// TwinCAT 3 PLC project PLCInterpolation
// libraries:
//   TC2_Converted,1.1.0.0,aaaa
//   Tc2_Math, * (Beckhoff Automation GmbH)
//   Tc2_NC, * (Beckhoff Automation GmbH)
//   Tc2_NCI, * (Beckhoff Automation GmbH)
//   Tc2_PlcInterpolation, * (Beckhoff Automation GmbH)
//   Tc2_Standard, * (Beckhoff Automation GmbH)
//   Tc2_System, * (Beckhoff Automation GmbH)
//   Tc2_Utilities, * (Beckhoff Automation GmbH)
//   Tc3_Module, * (Beckhoff Automation GmbH)
// project tree:
//   Data types/ E_ACTIONTYPE.TcDUT, E_CONTROL_MODE.TcDUT, E_PROGRAM_STATE.TcDUT, ST_EXECUTION_TABLE.TcDUT, ST_PROGRAM.TcDUT
//   Global Variables/ Global_Variables.TcGVL, PROGRAMS.TcGVL, SETTINGS.TcGVL, TwinCAT_Import.TcGVL, Variable_Configuration.TcGVL
//   POUs/ FB_AxisEnable.TcPOU, FB_ChannelReset.TcPOU, FB_ChannelStartStop.TcPOU, FB_Execute.TcPOU, FB_SelectProgram.TcPOU, MAIN.TcPOU
//   / Standard.TcTTO

CONFIGURATION PLCInterpolation
    RESOURCE PLC ON TwinCAT3
        TASK Standard(INTERVAL := T#10ms, PRIORITY := 22);
        PROGRAM MAIN WITH Standard : MAIN;
    END_RESOURCE
END_CONFIGURATION

// ---- Data types/E_ACTIONTYPE.TcDUT
TYPE E_ACTIONTYPE :
(
	NONE,
	MOVE_X,
	MOVE_Y,
	MOVE_XY,
	MOVE_CIRCULAR,
	HOME,
	END
);
END_TYPE

// ---- Data types/E_CONTROL_MODE.TcDUT
TYPE E_CONTROL_MODE :
(
	E_REF_MODE,
	E_JOG_MODE,
	E_AUTO_MODE
);
END_TYPE

// ---- Data types/E_PROGRAM_STATE.TcDUT
TYPE E_PROGRAM_STATE :
(
	E_PROGRAMSTATE_NONE,
	E_PROGRAMSTATE_READY,
	E_PROGRAMSTATE_RESETTED,
	E_PROGRAMSTATE_RUNNING,
	E_PROGRAMSTATE_STOPPED,
	E_PROGRAMSTATE_ERROR
);
END_TYPE

// ---- Data types/ST_EXECUTION_TABLE.TcDUT
TYPE ST_EXECUTION_TABLE :
STRUCT
	ActionType:E_ACTIONTYPE;
	X:LREAL;
	Y:LREAL;
	I:LREAL;
	J:LREAL;
	Clockwise:BOOL;
END_STRUCT
END_TYPE

// ---- Data types/ST_PROGRAM.TcDUT
TYPE ST_PROGRAM :
STRUCT
	Name:STRING;
	Comment:STRING;
	ExecutionTable:ARRAY[1..MAX_NUMBER_OF_TABLE_LINES] OF ST_EXECUTION_TABLE;
END_STRUCT
END_TYPE

// ---- Global Variables/Global_Variables.TcGVL
{attribute 'Tc2GvlVarNames'}
VAR_GLOBAL
	in_stXNcToPlc		AT %I*:	NCTOPLC_AXIS_REF;
	in_stYNcToPlc		AT %I*:	NCTOPLC_AXIS_REF;
	in_stZNcToPlc		AT %I*:	NCTOPLC_AXIS_REF;

	in_stItpToPlc		AT %I*:	NCTOPLC_NCICHANNEL_REF;


	out_stXPlcToNc		AT	%Q*:	PLCTONC_AXIS_REF;
	out_stYPlcToNc		AT	%Q*:	PLCTONC_AXIS_REF;
	out_stZPlcToNc		AT	%Q*:	PLCTONC_AXIS_REF;

	out_stPlcToItp		AT	%Q*:	PLCTONC_NCICHANNEL_REF;


	gGlobalEnable: BOOL:=TRUE;
	gFeedOverride:	LREAL	:= 100.0;
	gVelocity: UINT:=1000;

	gControlMode:E_CONTROL_MODE:=E_AUTO_MODE;			(* Defines is control in REF, JOG or AUTO mode *)
	gProgramState: E_PROGRAM_STATE;		(* Defines status of the current program *)
	gStatistics_LastProgramTime:REAL; (* Last program time in seconds *)


	(* Visualization variables *)
	gVisuStart:BOOL;
	gVisuStop:BOOL;
	gVisuReset:BOOL;

	gVisuPrgNumber: INT;
	gVisuSelectPrg: BOOL;

END_VAR

VAR_GLOBAL CONSTANT
	ItpChnId:	UDINT := 2;
	ItpGrpId:	UDINT := 4;

	MAX_NUMBER_OF_TABLE_LINES:UINT:=100;
	MAX_NUMBER_OF_PROGRAMS:UINT:=10;

END_VAR

// ---- Global Variables/PROGRAMS.TcGVL
{attribute 'Tc2GvlVarNames'}
VAR_GLOBAL PERSISTENT
	gPrograms:ARRAY[1..MAX_NUMBER_OF_PROGRAMS] OF ST_PROGRAM;
	gCurrentProgram:ST_PROGRAM;
	giProgramNumber:INT;
END_VAR

// ---- Global Variables/SETTINGS.TcGVL
{attribute 'Tc2GvlVarNames'}
VAR_GLOBAL PERSISTENT
	(* Axis reference positions *)
	X_REF:LREAL:=0;
	Y_REF:LREAL:=0;

	(* Home position for axis *)
	X_Home:LREAL:=0;
	Y_Home:LREAL:=0;

END_VAR

// ---- Global Variables/TwinCAT_Import.TcGVL
{attribute 'Tc2GvlVarNames'}
(* Generated automatically by TwinCAT - do not edit manually! *)
VAR_GLOBAL
END_VAR

// ---- Global Variables/Variable_Configuration.TcGVL
{attribute 'Tc2GvlVarNames'}
VAR_CONFIG
END_VAR

// ---- POUs/MAIN.TcPOU
PROGRAM MAIN
VAR
	fbBuilGroup: CfgBuildExt3DGroup;
	fbExecute: FB_Execute;
	fbChannelReset: FB_ChannelReset;

	fbStartStop: FB_ChannelStartStop;
	rtSlideStart:R_TRIG;

	tmrReset: TON;

	fbSelectPrg: FB_SelectProgram;

	fbReleaseGroup: CfgReconfigGroup;

	fbEnable: FB_AxisEnable;
END_VAR

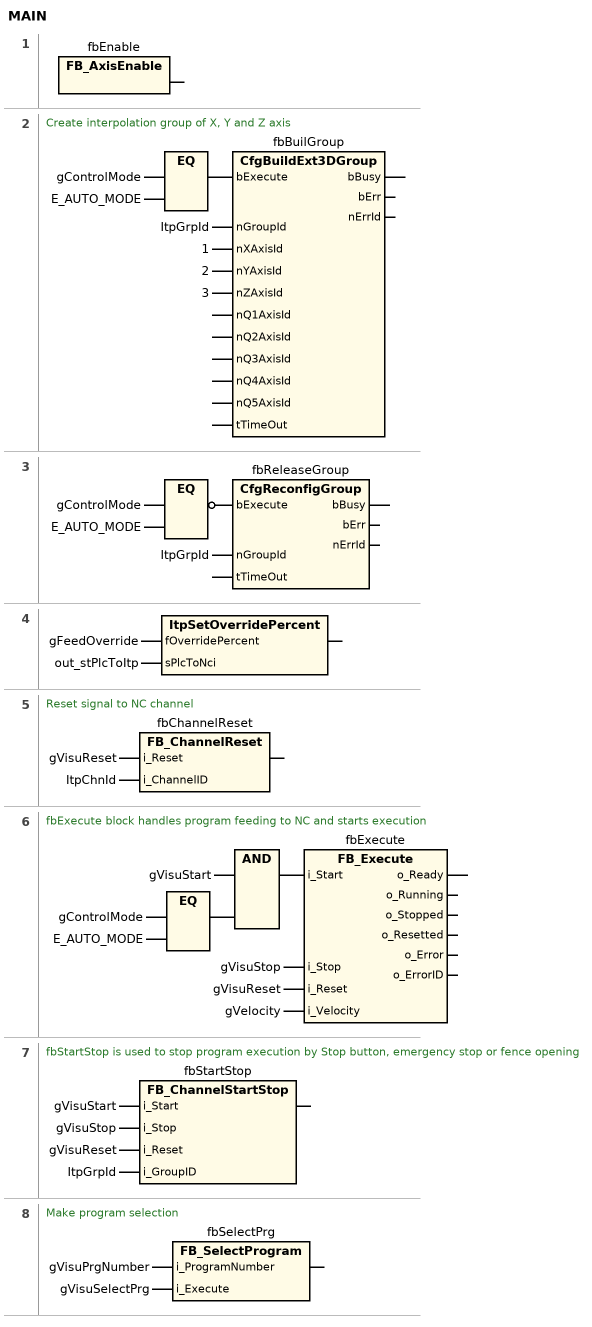
// NETWORK 1
fbEnable(); // FB_AxisEnable

// NETWORK 2
// Create interpolation group of X, Y and Z axis
fbBuilGroup(
    bExecute := gControlMode = E_AUTO_MODE,
    nGroupId := ItpGrpId,
    nXAxisId := 1,
    nYAxisId := 2,
    nZAxisId := 3); // CfgBuildExt3DGroup

// NETWORK 3
fbReleaseGroup(bExecute := NOT (gControlMode = E_AUTO_MODE), nGroupId := ItpGrpId); // CfgReconfigGroup

// NETWORK 4
ItpSetOverridePercent(fOverridePercent := gFeedOverride, sPlcToNci := out_stPlcToItp);

// NETWORK 5
// Reset signal to NC channel
fbChannelReset(i_Reset := gVisuReset, i_ChannelID := ItpChnId); // FB_ChannelReset

// NETWORK 6
// fbExecute block handles program feeding to NC and starts execution
fbExecute(
    i_Start := gVisuStart AND gControlMode = E_AUTO_MODE,
    i_Stop := gVisuStop,
    i_Reset := gVisuReset,
    i_Velocity := gVelocity); // FB_Execute

// NETWORK 7
// fbStartStop is used to stop program execution by Stop button, emergency stop or fence opening
fbStartStop(i_Start := gVisuStart, i_Stop := gVisuStop, i_Reset := gVisuReset, i_GroupID := ItpGrpId); // FB_ChannelStartStop

// NETWORK 8
// Make program selection
fbSelectPrg(i_ProgramNumber := gVisuPrgNumber, i_Execute := gVisuSelectPrg); // FB_SelectProgram

END_PROGRAM

// ---- POUs/FB_Execute.TcPOU
FUNCTION_BLOCK FB_Execute
VAR_INPUT
	i_Start:BOOL;
	i_Stop:BOOL;
	i_Reset:BOOL;
	i_Velocity: UINT;
END_VAR
VAR_OUTPUT
	o_Ready:BOOL;
	o_Running:BOOL;
	o_Stopped:BOOL;
	o_Resetted:BOOL;
	o_Error:BOOL;
	o_ErrorID:DINT;
END_VAR
VAR
	(* test feeding 10 lines at time *)
	bFeedMore:BOOL;

	iProgramLine:UINT:=1;
	oldStart: BOOL;

	stNciFeedGroupTable:	ST_NciFeedGroupTable;
	fbFeedTablePrep:FB_NciFeedTablePreparation;
	stGeoStart:ST_NciGeoStart;
	stGeoLine:ST_NciGeoLine;
	stGeoCirclePlane:	ST_NciGeoCirclePlane;
	stEndOfTables:	ST_NciEndOfTables;
	stMFuncHsk:ST_NciMFuncHsk;
	nFilledRows:	UDINT	:= 0;
	bError:	BOOL	:= FALSE;
	nErrorId:	UDINT := 0;
	fbFeedTable:FB_NciFeedTable;


	bFeed: BOOL;
	lPreviousX:LREAL;
	lPreviousY:LREAL;
	bEnd: BOOL;
	nEndStep: INT;
	tmrProgramTime: TON;
END_VAR

IF i_Start AND NOT oldStart AND ((gProgramState=E_PROGRAMSTATE_RESETTED) OR (gProgramState=E_PROGRAMSTATE_READY) OR (gProgramState=E_PROGRAMSTATE_NONE)) THEN
	iProgramLine:=1;
	gProgramState:=E_PROGRAMSTATE_RUNNING;
	bEnd:=FALSE;
	nEndStep:=0;
	o_Ready:=FALSE;

	(* GeoStart is required if the first geo entry is a circle is first used movement *)
	(* Take current position as start position *)
	stGeoStart.fPosX:= lPreviousX:=in_stXNcToPlc.ActPos;
	stGeoStart.fPosY:= lPreviousY:=in_stYNcToPlc.ActPos;

	fbFeedTablePrep(
		nEntryType:= E_NciEntryTypeGeoStart,
		pEntry:= ADR(stGeoStart) ,
		bResetTable:= FALSE,
		bResetAll:=FALSE,
		stFeedGroupTable:= stNciFeedGroupTable,
		nFilledRows=>nFilledRows,
		bError=>bError,
		nErrorId=> nErrorId);
END_IF

oldStart:=i_Start;

IF (gProgramState=E_PROGRAMSTATE_RUNNING) AND i_Stop THEN
	gProgramState:=E_PROGRAMSTATE_STOPPED;
END_IF
IF (gProgramState=E_PROGRAMSTATE_STOPPED) AND i_Start THEN
	gProgramState:=E_PROGRAMSTATE_RUNNING;
END_IF


IF i_Reset THEN
	bEnd:=FALSE;
	nEndStep:=0;
	bFeed:=FALSE;
	o_Error:=FALSE;
	o_ErrorID:=0;
	o_Ready:=FALSE;
	gProgramState:=E_PROGRAMSTATE_RESETTED;
	iProgramLine:=1;
	fbFeedTablePrep(
		bResetAll:= TRUE,
		stFeedGroupTable:= stNciFeedGroupTable);
	fbFeedTable.bExecute := FALSE;
END_IF

IF gProgramState=E_PROGRAMSTATE_RUNNING AND (NOT bEnd) THEN
	CASE gCurrentProgram.ExecutionTable[iProgramLine].ActionType OF
		MOVE_X:
			stGeoLine.nDisplayIndex	:= iProgramLine;
			stGeoLine.fEndPosX	:=lPreviousX:=gCurrentProgram.ExecutionTable[iProgramLine].X;
			stGeoLine.fEndPosY:= lPreviousY;
			stGeoLine.fVelo		:= i_Velocity; (*mm per sec*)

			fbFeedTablePrep(
				nEntryType:= E_NciEntryTypeGeoLine,
				pEntry:= ADR(stGeoLine),
				bResetTable:= FALSE,
				stFeedGroupTable:= stNciFeedGroupTable,
				nFilledRows=>nFilledRows,
				bError=>bError,
				nErrorId=> nErrorId);

			iProgramLine:=iProgramLine+1;

		MOVE_Y:
			stGeoLine.nDisplayIndex	:= iProgramLine;
			stGeoLine.fEndPosX	:= lPreviousX;
			stGeoLine.fEndPosY:=lPreviousY:=gCurrentProgram.ExecutionTable[iProgramLine].Y;
			stGeoLine.fVelo		:= i_Velocity; (*mm per sec*)

			fbFeedTablePrep(
				nEntryType:= E_NciEntryTypeGeoLine,
				pEntry:= ADR(stGeoLine),
				bResetTable:= FALSE,
				stFeedGroupTable:= stNciFeedGroupTable,
				nFilledRows=>nFilledRows,
				bError=>bError,
				nErrorId=> nErrorId);

			iProgramLine:=iProgramLine+1;

		MOVE_XY:
			stGeoLine.nDisplayIndex	:= iProgramLine;
			stGeoLine.fEndPosX	:=lPreviousX:=gCurrentProgram.ExecutionTable[iProgramLine].X;
			stGeoLine.fEndPosY:= lPreviousY:=gCurrentProgram.ExecutionTable[iProgramLine].Y;
			stGeoLine.fVelo		:= i_Velocity; (*mm per sec*)

			fbFeedTablePrep(
				nEntryType:= E_NciEntryTypeGeoLine,
				pEntry:= ADR(stGeoLine),
				bResetTable:= FALSE,
				stFeedGroupTable:= stNciFeedGroupTable,
				nFilledRows=>nFilledRows,
				bError=>bError,
				nErrorId=> nErrorId);

			iProgramLine:=iProgramLine+1;

		MOVE_CIRCULAR:
			stGeoCirclePlane.nDisplayIndex	:= iProgramLine;
			stGeoCirclePlane.fEndPosX	:= lPreviousX:=gCurrentProgram.ExecutionTable[iProgramLine].X;
			stGeoCirclePlane.fEndPosY	:= lPreviousY:=gCurrentProgram.ExecutionTable[iProgramLine].Y;
			stGeoCirclePlane.fCenterX	:= gCurrentProgram.ExecutionTable[iProgramLine].I;
			stGeoCirclePlane.fCenterY	:= gCurrentProgram.ExecutionTable[iProgramLine].J;
			stGeoCirclePlane.fVelo	:= i_Velocity; (*mm per sec*)
			stGeoCirclePlane.bClockwise	:= gCurrentProgram.ExecutionTable[iProgramLine].Clockwise;

			fbFeedTablePrep(
				nEntryType:= E_NciEntryTypeGeoCirclePlane,
				pEntry:= ADR(stGeoCirclePlane),
				bResetTable:= FALSE,
				stFeedGroupTable:= stNciFeedGroupTable,
				nFilledRows=>nFilledRows,
				bError=>bError,
				nErrorId=> nErrorId);

			iProgramLine:=iProgramLine+1;

		HOME:
			(* X Axis to home position *)
			stGeoLine.nDisplayIndex	:= iProgramLine;
			stGeoLine.fEndPosX	:=lPreviousX:=X_Home;
			stGeoLine.fEndPosY:= lPreviousY;
			stGeoLine.fVelo		:= i_Velocity; (*mm per sec*)

			fbFeedTablePrep(
				nEntryType:= E_NciEntryTypeGeoLine,
				pEntry:= ADR(stGeoLine),
				bResetTable:= FALSE,
				stFeedGroupTable:= stNciFeedGroupTable,
				nFilledRows=>nFilledRows,
				bError=>bError,
				nErrorId=> nErrorId);

			(* Y Axis to home position *)
			stGeoLine.nDisplayIndex	:= iProgramLine;
			stGeoLine.fEndPosX	:= lPreviousX;
			stGeoLine.fEndPosY:=Y_Home;
			stGeoLine.fVelo		:= i_Velocity; (*mm per sec*)

			fbFeedTablePrep(
				nEntryType:= E_NciEntryTypeGeoLine,
				pEntry:= ADR(stGeoLine),
				bResetTable:= FALSE,
				stFeedGroupTable:= stNciFeedGroupTable,
				nFilledRows=>nFilledRows,
				bError=>bError,
				nErrorId=> nErrorId);

			iProgramLine:=iProgramLine+1;

		END:
			bEnd:=TRUE;
			(* End of movements *)
			fbFeedTablePrep(
				nEntryType:= E_NciEntryTypeEndOfTables,
				pEntry:= ADR(stEndOfTables),
				bResetTable:= FALSE,
				stFeedGroupTable:= stNciFeedGroupTable,
				nFilledRows=>nFilledRows,
				bError=>bError,
				nErrorId=> nErrorId);
			nEndStep:=10;

	END_CASE
END_IF

IF bEnd THEN
	CASE nEndStep OF
		10:
			(* write data down to NC kernel *)
			fbFeedTable.bExecute:= TRUE;
			nEndStep:=20;

		20:
			IF fbFeedTable.bFeedingDone THEN
				fbFeedTablePrep(
					bResetAll:= TRUE,
					stFeedGroupTable:= stNciFeedGroupTable);

				fbFeedTable.bExecute:= FALSE;
				nEndStep:=30;
			END_IF
		30:	(* Wait for program ready *)

			IF fbFeedTable.bChannelDone THEN
				nEndStep:=40;
			END_IF

		40:

				o_Ready:=TRUE;
				o_Running:=FALSE;
				gProgramState:=E_PROGRAMSTATE_READY;
				gStatistics_LastProgramTime:=TIME_TO_REAL( tmrProgramTime.ET)/100;
				nEndStep:=0;
	END_CASE
END_IF

fbFeedTable(
	stFeedGroupTable:= stNciFeedGroupTable,
	stNciToPlc:=  in_stItpToPlc);


tmrProgramTime(IN:=(gProgramState=E_PROGRAMSTATE_RUNNING),PT:=T#100S);

END_FUNCTION_BLOCK

// ---- POUs/FB_ChannelReset.TcPOU
FUNCTION_BLOCK FB_ChannelReset

VAR_INPUT
	i_Reset:BOOL;
	i_ChannelID: UDINT;

END_VAR
VAR_OUTPUT
END_VAR
VAR
	fbReset: ItpReset;
END_VAR

fbReset(
	bExecute:= i_Reset,
	nChnId:= i_ChannelID,
	tTimeOut:= T#1S,
	bBusy=> ,
	bErr=> ,
	nErrId=> );

END_FUNCTION_BLOCK

// ---- POUs/FB_ChannelStartStop.TcPOU
FUNCTION_BLOCK FB_ChannelStartStop
VAR_INPUT
	i_Start:BOOL;
	i_Stop:BOOL;
	i_Reset:BOOL;
	i_GroupID:UDINT;
END_VAR
VAR_OUTPUT
END_VAR
VAR
	bStopped:BOOL;

	fbItpStepOnAfterEStop: ItpStepOnAfterEStop;
	fbItpEStop: ItpEStop;
END_VAR

fbItpStepOnAfterEStop(
	bExecute:= i_Start AND bStopped,
	nGrpId:=i_GroupID ,
	tTimeOut:= t#1S,
	bBusy=> ,
	bErr=> ,
	nErrId=> );

fbItpEStop(
	bExecute:=i_Stop ,
	nGrpId:= i_GroupID,
	fDec:= 10000,
	fJerk:= 1000000,
	tTimeOut:= T#1S,
	bBusy=> ,
	bErr=> ,
	nErrId=> );

IF i_Stop THEN
	bStopped:=TRUE;
END_IF

IF i_Reset THEN
	bStopped := FALSE;
END_IF

END_FUNCTION_BLOCK

// ---- POUs/FB_SelectProgram.TcPOU
FUNCTION_BLOCK FB_SelectProgram
VAR_INPUT
	i_ProgramNumber:UINT;
	i_Execute:BOOL;
END_VAR
VAR
	oldExecute: BOOL;
END_VAR

(* Check that program number is within valid range *)
IF i_Execute AND NOT oldExecute THEN
	gCurrentProgram := gPrograms[i_ProgramNumber];
	giProgramNumber:=i_ProgramNumber;
END_IF
oldExecute:=i_Execute;

END_FUNCTION_BLOCK

// ---- POUs/FB_AxisEnable.TcPOU
FUNCTION_BLOCK FB_AxisEnable
VAR_INPUT
END_VAR
VAR_OUTPUT
END_VAR
VAR
	fbXAxis: MC_Power;
	fbYAxis: MC_Power;
	fbZAxis: MC_Power;
END_VAR

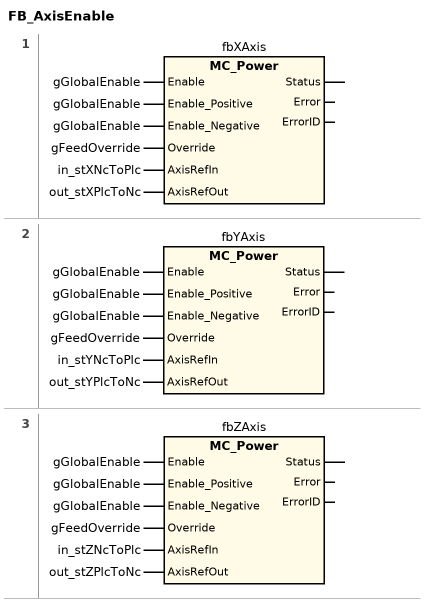
// NETWORK 1
fbXAxis(
    Enable := gGlobalEnable,
    Enable_Positive := gGlobalEnable,
    Enable_Negative := gGlobalEnable,
    Override := gFeedOverride,
    AxisRefIn := in_stXNcToPlc,
    AxisRefOut := out_stXPlcToNc); // MC_Power

// NETWORK 2
fbYAxis(
    Enable := gGlobalEnable,
    Enable_Positive := gGlobalEnable,
    Enable_Negative := gGlobalEnable,
    Override := gFeedOverride,
    AxisRefIn := in_stYNcToPlc,
    AxisRefOut := out_stYPlcToNc); // MC_Power

// NETWORK 3
fbZAxis(
    Enable := gGlobalEnable,
    Enable_Positive := gGlobalEnable,
    Enable_Negative := gGlobalEnable,
    Override := gFeedOverride,
    AxisRefIn := in_stZNcToPlc,
    AxisRefOut := out_stZPlcToNc); // MC_Power

END_FUNCTION_BLOCK
